// TwinCAT 3 PLC project mobject_collections
// Title: mobject-collections
// Company: mobject
// Author: mobject dev team
// ProjectVersion: 1.2.0
// ProgramVersion: 3.1.4023.0
// libraries:
//   mobject-disposable, * (mobject)
//   mobject-enumerable, * (mobject)
//   mobject-events, * (mobject)
//   Tc2_System, * (Beckhoff Automation GmbH)
//   Tc3_DynamicMemory, * (Beckhoff Automation GmbH)
// project tree:
//   Dictionary/ Dictionary.TcPOU (not stored)
//   Interfaces/Collections/Events/ I_CollectionChangedEvent.TcIO (not stored), I_CollectionDisposedEvent.TcIO (not stored)
//   Interfaces/Collections/ I_Collection.TcIO (not stored), I_List.TcIO (not stored), I_LinkedList.TcIO (not stored), I_Queue.TcIO (not stored), I_Stack.TcIO (not stored)
//   Interfaces/Collections/Nodes/ I_CollectionNode.TcIO (not stored), I_LinkedListNode.TcIO (not stored), I_ListNode.TcIO (not stored)
//   Interfaces/KeyValueCollections/Events/ I_KeyValueCollectionChangedEvent.TcIO (not stored), I_KeyValueCollectionDisposedEvent.TcIO (not stored)
//   Interfaces/KeyValueCollections/ I_Dictionary.TcIO (not stored), I_KeyValueCollection.TcIO (not stored)
//   Interfaces/KeyValueCollections/Nodes/ I_DictionaryTreeNode.TcIO (not stored), I_OrderedDictionaryTreeNode.TcIO (not stored)
//   LinkedList/ LinkedList.TcPOU (not stored)
//   List/ List.TcPOU
//   OrderedDictionary/ OrderedDictionary.TcPOU (not stored)
//   Queue/ Queue.TcPOU (not stored)
//   Stack/ Stack.TcPOU (not stored)
//   _Internal/Dictionary/Enumerator/ DictionaryForwardEnumerator.TcPOU (not stored)
//   _Internal/Dictionary/Node/ DictionaryTreeNode.TcPOU (not stored)
//   _Internal/Events/Collection/ CollectionChangedEvent.TcPOU (not stored), CollectionDisposedEvent.TcPOU (not stored), CollectionEvent.TcPOU (not stored)
//   _Internal/Events/KeyValueCollection/ KeyValueCollectionChangedEvent.TcPOU (not stored), KeyValueCollectionDisposedEvent.TcPOU (not stored), KeyValueCollectionEvent.TcPOU (not stored)
//   _Internal/LinkedList/Enumerator/ LinkedListForwardEnumerator.TcPOU (not stored)
//   _Internal/LinkedList/Node/ LinkedListNode.TcPOU (not stored)
//   _Internal/List/Enumerator/ ListForwardEnumerator.TcPOU (not stored)
//   _Internal/List/Node/ ListNode.TcPOU (not stored)
//   _Internal/OrderedDictionary/Enumerator/ OrderedDictionaryForwardEnumerator.TcPOU (not stored)
//   _Internal/OrderedDictionary/Node/ OrderedDictionaryTreeNode.TcPOU (not stored)

// ---- List/List.TcPOU
{attribute 'linkalways'} 
{attribute 'no_explicit_call' := 'This FB is a CLASS and must be accessed using methods or properties'}
{attribute 'enable_dynamic_creation'}
{attribute 'hide_all_locals'}
FUNCTION_BLOCK PUBLIC List EXTENDS Disposable IMPLEMENTS I_List
VAR
	memoryManager : FB_DynMem_Manager2;
	buffer : FB_DynMem_Buffer(ipMemMan := memoryManager);
	pArrayOfListNodes : POINTER TO I_ListNode;
	arrayCapacity : DINT;
	itemCount : DINT;
	eventEmitter : EventEmitter;
END_VAR

METHOD PUBLIC AddItem
VAR_INPUT
	Item : ANY;
END_VAR
VAR
	node : I_ListNode;
END_VAR
node := CreateNewNode(Item);
IF AddNodeLast(node) THEN
	EmitChangedEvent();
END_IF
END_METHOD

METHOD PRIVATE AddNodeAt : BOOL
VAR_INPUT
	Index : DINT;
	Node : I_ListNode;
END_VAR
VAR
	i : DINT;
END_VAR
IF Index = itemCount THEN
	IF AddNodeLast(Node) THEN
		AddNodeAt := TRUE;
	END_IF
	RETURN;
END_IF

IF Index > itemCount - 1 THEN
	RETURN;
END_IF

IF itemCount + 1 > arrayCapacity THEN
	IF NOT Grow() THEN
		RETURN;
	END_IF
END_IF

IF IsBufferPointerValid THEN
	//Move all excisting nodes up
	FOR i := itemCount - 1 TO Index BY -1 DO
		pArrayOfListNodes[i + 1] := pArrayOfListNodes[i];
		pArrayOfListNodes[i] := 0;
	END_FOR
	
	pArrayOfListNodes[Index] := Node;
	itemCount := itemCount + 1;
	
	AddNodeAt := TRUE;
END_IF
END_METHOD

METHOD PRIVATE AddNodeLast : BOOL
VAR_INPUT
	Node : I_ListNode;
END_VAR
IF itemCount = arrayCapacity THEN
    IF NOT Grow() THEN
		RETURN;
	END_IF
END_IF

IF IsBufferPointerValid THEN
	pArrayOfListNodes[itemCount] := Node;
	itemCount := itemCount + 1;
	
	AddNodeLast := TRUE;
END_IF
END_METHOD

PROPERTY PUBLIC Capacity : DINT
GET
Capacity := arrayCapacity;
END_GET
END_PROPERTY

METHOD Clear
VAR_INPUT
END_VAR
IF IsEmpty THEN
	RETURN;
END_IF

RemoveAllNodes();
EmitChangedEvent();
END_METHOD

METHOD Contains : BOOL
VAR_INPUT
	Item : ANY;
END_VAR
IF IsEmpty THEN
	RETURN;
END_IF

Contains := GetIndexOf(Item) > -1;
END_METHOD

PROPERTY PUBLIC Count : DINT
GET
Count := itemCount;
END_GET
END_PROPERTY

METHOD PRIVATE CreateNewNode : I_ListNode
VAR_INPUT
	Value : ANY;
END_VAR
VAR
	pNode : POINTER TO ListNode;
END_VAR
pNode := __NEW(ListNode(Source := Value));
CreateNewNode := pNode^;
END_METHOD

METHOD PRIVATE EmitChangedEvent
VAR
	pCollectionChangedEvent : POINTER TO CollectionChangedEvent;
END_VAR
pCollectionChangedEvent := __NEW(CollectionChangedEvent(Target := THIS^));
eventEmitter.Emit('OnChanged', pCollectionChangedEvent^);
pCollectionChangedEvent^.Dispose();
END_METHOD

METHOD PRIVATE EmitDisposedEvent
VAR
	pCollectionDisposedEvent : POINTER TO CollectionDisposedEvent;
END_VAR
pCollectionDisposedEvent := __NEW(CollectionDisposedEvent(Target := THIS^));
eventEmitter.Emit('OnDisposed', pCollectionDisposedEvent^);
pCollectionDisposedEvent^.Dispose();
END_METHOD

METHOD FB_exit : BOOL
VAR_INPUT
	bInCopyCode : BOOL; // if TRUE, the exit method is called for exiting an instance that is copied afterwards (online change).
END_VAR
VAR
END_VAR
IF bInCopyCode THEN
    RETURN;
END_IF

Clear();
buffer.DeleteBuffer();
EmitDisposedEvent();
END_METHOD

METHOD GetEnumerator : I_ForwardEnumerator
VAR
	pEnumerator : POINTER TO ListForwardEnumerator;
END_VAR
pEnumerator := __NEW(ListForwardEnumerator(Parent := THIS^));
GetEnumerator := pEnumerator^;
END_METHOD

METHOD PUBLIC GetIndexOf : DINT
VAR_INPUT
	Item : ANY;
END_VAR
VAR
	node : I_ListNode;
	i : DINT;
END_VAR
GetIndexOf := -1;

IF IsEmpty THEN
	RETURN;
END_IF

FOR i := 0 TO itemCount - 1 DO
	node := THIS^.GetItemAtIndex(i);
	
	IF node.Equals(Item) THEN
		GetIndexOf := i;
		RETURN;
	END_IF
END_FOR
END_METHOD

METHOD PRIVATE GetItemAtIndex : I_ListNode
VAR_INPUT
	Index : DINT;
END_VAR
IF IsNotValidIndex(Index) THEN
	RETURN;
END_IF

IF IsBufferPointerValid THEN
	GetItemAtIndex := pArrayOfListNodes[Index];
END_IF
END_METHOD

METHOD PRIVATE Grow : BOOL
VAR
	node : I_ListNode;
	
	nodeSize: UINT;
	creationSize: UDINT;
	bufferTemp: PVOID;
END_VAR
VAR CONSTANT
    INITIAL_CAPACITY : DINT := 4;
END_VAR
IF arrayCapacity = 0 THEN
	arrayCapacity := INITIAL_CAPACITY;
ELSE
	arrayCapacity := arrayCapacity * 2;
END_IF

nodeSize := SIZEOF(node);
creationSize := DINT_TO_UDINT(arrayCapacity) * nodeSize;
bufferTemp := buffer.pBuffer;

buffer.CreateBuffer(nSize := 512, bReset := TRUE);
bufferTemp := buffer.pBuffer;

IF buffer.bAvailable THEN
	IF NOT buffer.Resize(nSize := DINT_TO_UDINT(arrayCapacity) * SIZEOF(node), bPreserve := TRUE, bReset := FALSE) THEN
		RETURN;
	END_IF
ELSE
	IF NOT buffer.CreateBuffer(nSize := DINT_TO_UDINT(arrayCapacity) * SIZEOF(node), bReset := TRUE) THEN
		RETURN;
	END_IF
END_IF

IF buffer.bAvailable THEN
	pArrayOfListNodes := buffer.pBuffer;
	
	IF IsBufferPointerValid THEN
		Grow := TRUE;
	END_IF
END_IF
END_METHOD

PROPERTY PRIVATE IsBufferPointerValid : BOOL
GET
IsBufferPointerValid := pArrayOfListNodes <> 0;
END_GET
END_PROPERTY

PROPERTY IsEmpty : BOOL
GET
IsEmpty := itemCount = 0;
END_GET
END_PROPERTY

METHOD PRIVATE IsNotValidIndex : BOOL
VAR_INPUT
	Index : DINT;
END_VAR
IsNotValidIndex := NOT IsValidIndex(Index);
END_METHOD

METHOD PRIVATE IsValidIndex : BOOL
VAR_INPUT
	Index : DINT;
END_VAR
IF Index < 0 THEN
	RETURN;
END_IF

IF Index >= itemCount THEN
	RETURN;
END_IF

IsValidIndex := TRUE;
END_METHOD

METHOD PUBLIC OffEvent
VAR_INPUT
	EventName : T_MaxString;
	EventHandler : I_EventHandler;
END_VAR
eventEmitter.OffEvent(EventName, EventHandler);
END_METHOD

METHOD PUBLIC OnceEvent
VAR_INPUT
	EventName : T_MaxString;
	EventHandler : I_EventHandler;
END_VAR
eventEmitter.OnceEvent(EventName, EventHandler);
END_METHOD

METHOD PUBLIC OnEvent
VAR_INPUT
	EventName : T_MaxString;
	EventHandler : I_EventHandler;
END_VAR
eventEmitter.OnEvent(EventName, EventHandler);
END_METHOD

METHOD PRIVATE RemoveAllNodes
VAR
	i : DINT;
END_VAR
FOR i := 0 TO itemCount - 1 DO
	IF pArrayOfListNodes[i] <> 0 THEN
		pArrayOfListNodes[i].Dispose();
	END_IF
END_FOR

itemCount := 0;
END_METHOD

METHOD PUBLIC TrimExcess
VAR
	node : I_ListNode;
END_VAR
IF arrayCapacity = 0 THEN
	RETURN;
END_IF

IF arrayCapacity = itemCount THEN
	RETURN;
END_IF

arrayCapacity := itemCount;
IF buffer.Resize(nSize := DINT_TO_UDINT(arrayCapacity) * SIZEOF(node), bPreserve := TRUE, bReset := FALSE) THEN
	pArrayOfListNodes := buffer.pBuffer;
ELSE
	pArrayOfListNodes := 0;
END_IF
END_METHOD

METHOD PUBLIC TryCopyTo : BOOL
VAR_INPUT
	Destination	: ANY;
END_VAR
TryCopyTo := TryCopyToLocation(Destination.pValue, DINT_TO_UDINT(Destination.diSize));
END_METHOD

METHOD PUBLIC TryCopyToLocation : BOOL
VAR_INPUT
	DestinationAddress : PVOID;
	DestinationSize : UDINT;
END_VAR
VAR
	i : DINT;
	requiredSize : UDINT;
	current : I_ListNode;
	pCurrent : PVOID;
END_VAR
IF IsEmpty THEN
    RETURN;
END_IF

//Compute required size
FOR i := 0 TO Count - 1 DO
    current := GetItemAtIndex(i);
    requiredSize := requiredSize + current.DataSize;
END_FOR

//If destination size is to small abort
IF DestinationSize < requiredSize THEN
    RETURN;
END_IF

pCurrent := DestinationAddress;

FOR i := 0 TO Count - 1 DO
    current := GetItemAtIndex(i);
    current.TryGetTo(pCurrent, current.DataSize);
    pCurrent := pCurrent + current.DataSize;
END_FOR
END_METHOD

METHOD PUBLIC TryGetByIndex : BOOL
VAR_INPUT
	Index : DINT;
	Destination : ANY;
END_VAR
VAR
	node : I_ListNode;
END_VAR
node := GetItemAtIndex(Index);

IF node = 0 THEN
	RETURN;
END_IF

TryGetByIndex := node.TryGet(Destination);
END_METHOD

METHOD PUBLIC TryGetToByIndex : BOOL
VAR_INPUT
	Index : DINT;
	DestinationAddress : PVOID;
	DestinationSize : UDINT;
END_VAR
VAR
	node : I_ListNode;
END_VAR
node := GetItemAtIndex(Index);

IF node = 0 THEN
	RETURN;
END_IF

TryGetToByIndex := node.TryGetTo(DestinationAddress, DestinationSize);
END_METHOD

METHOD TryInsert : BOOL
VAR_INPUT
	Index : DINT;
	Item : ANY;
END_VAR
VAR
	node : I_ListNode;
END_VAR
IF IsNotValidIndex(Index) THEN
	RETURN;
END_IF

node := CreateNewNode(Item);
IF AddNodeAt(Index, node) THEN
	EmitChangedEvent();
	TryInsert := TRUE;
END_IF
END_METHOD

METHOD PUBLIC TryRemoveAt : BOOL;
VAR_INPUT
	Index : DINT;
END_VAR
VAR
	i : DINT;
	node : I_ListNode;
END_VAR
IF IsNotValidIndex(Index) THEN
	RETURN;
END_IF

IF IsBufferPointerValid THEN
	node := GetItemAtIndex(Index);
	node.Dispose();
	
	FOR i := Index + 1 TO itemCount - 1 DO
		pArrayOfListNodes[i - 1] := pArrayOfListNodes[i];
		pArrayOfListNodes[i] := 0;
	END_FOR
	
	itemCount := itemCount - 1;
	EmitChangedEvent();
	TryRemoveAt := TRUE;
END_IF
END_METHOD

METHOD TryRemoveItem : BOOL
VAR_INPUT
    Item : ANY;
END_VAR
VAR
    index : DINT;
END_VAR
index := GetIndexOf(Item);

IF index = -1 THEN
	RETURN;
END_IF

TryRemoveItem := TryRemoveAt(index);
END_METHOD

END_FUNCTION_BLOCK
